PROGRAM Module_Status
VAR
	BLINK_Check		: Blink;
	BLINK_Module	: Blink;
	Index			: INT;
	TimerModule		: ARRAY [1..10] OF TOF;
	Ethercat_Status : ARRAY [1..10] OF Ethercat_status;
	FB_SystemData	: SystemData;
	FB_CpuUsage		: TC_CpuUsage;
	FB_SysLatency	: TC_SysLatency;
	FB_UPS			: FB_S_UPS_CX51x0;
END_VAR

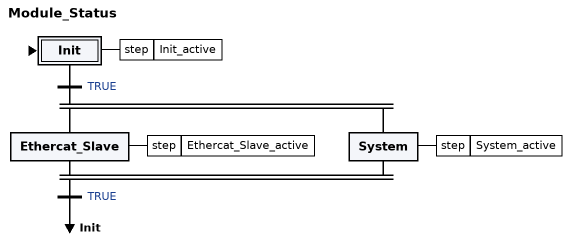
INITIAL_STEP Init:
    Init_active(N);  // step action
END_STEP
TRANSITION FROM Init TO (Ethercat_Slave, System)
    := TRUE;
END_TRANSITION
STEP Ethercat_Slave:
    Ethercat_Slave_active(N);  // step action
END_STEP
STEP System:
    System_active(N);  // step action
END_STEP
TRANSITION FROM (Ethercat_Slave, System) TO Init
    := TRUE;
END_TRANSITION

ACTION Ethercat_Slave_active:
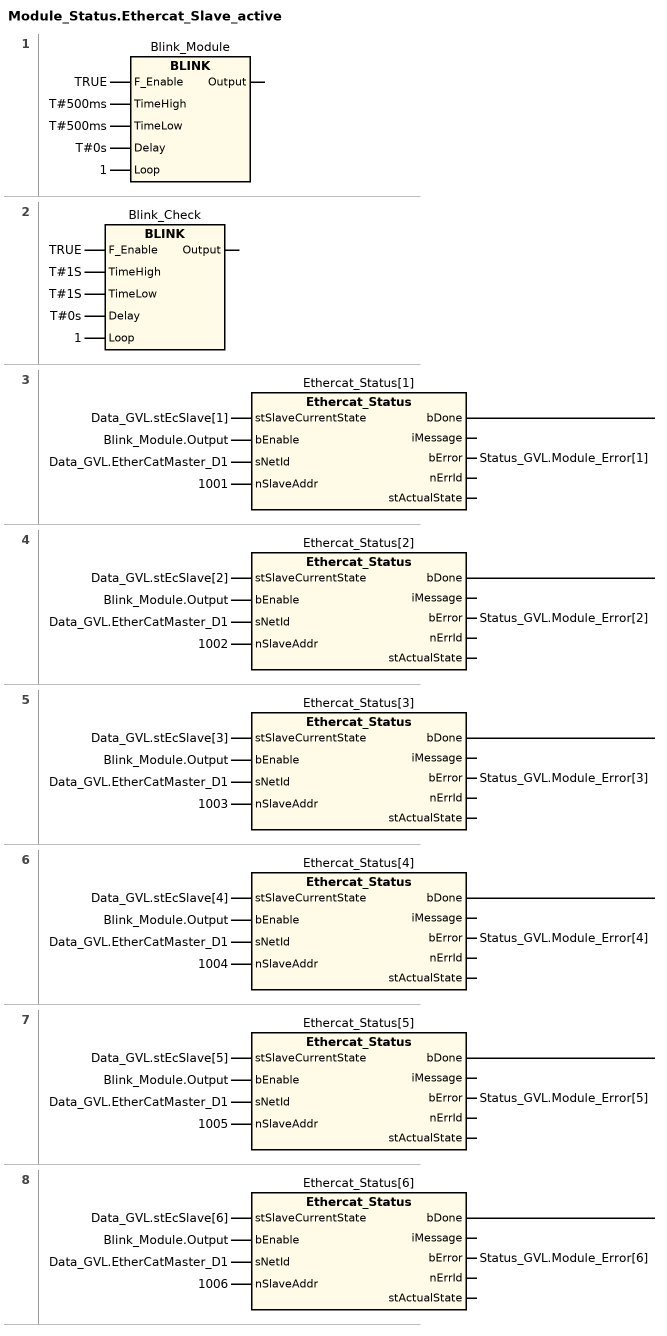
// NETWORK 1
Blink_Module(F_Enable := TRUE, TimeHigh := T#500ms, TimeLow := T#500ms, Delay := T#0s, Loop := 1); // BLINK

// NETWORK 2
Blink_Check(F_Enable := TRUE, TimeHigh := T#1S, TimeLow := T#1S, Delay := T#0s, Loop := 1); // BLINK

// NETWORK 3
Ethercat_Status[1](
    stSlaveCurrentState := Data_GVL.stEcSlave[1],
    bEnable := Blink_Module.Output,
    sNetId := Data_GVL.EtherCatMaster_D1,
    nSlaveAddr := 1001,
    bError => Status_GVL.Module_Error[1]); // Ethercat_Status

// NETWORK 4
Ethercat_Status[2](
    stSlaveCurrentState := Data_GVL.stEcSlave[2],
    bEnable := Blink_Module.Output,
    sNetId := Data_GVL.EtherCatMaster_D1,
    nSlaveAddr := 1002,
    bError => Status_GVL.Module_Error[2]); // Ethercat_Status

// NETWORK 5
Ethercat_Status[3](
    stSlaveCurrentState := Data_GVL.stEcSlave[3],
    bEnable := Blink_Module.Output,
    sNetId := Data_GVL.EtherCatMaster_D1,
    nSlaveAddr := 1003,
    bError => Status_GVL.Module_Error[3]); // Ethercat_Status

// NETWORK 6
Ethercat_Status[4](
    stSlaveCurrentState := Data_GVL.stEcSlave[4],
    bEnable := Blink_Module.Output,
    sNetId := Data_GVL.EtherCatMaster_D1,
    nSlaveAddr := 1004,
    bError => Status_GVL.Module_Error[4]); // Ethercat_Status

// NETWORK 7
Ethercat_Status[5](
    stSlaveCurrentState := Data_GVL.stEcSlave[5],
    bEnable := Blink_Module.Output,
    sNetId := Data_GVL.EtherCatMaster_D1,
    nSlaveAddr := 1005,
    bError => Status_GVL.Module_Error[5]); // Ethercat_Status

// NETWORK 8
Ethercat_Status[6](
    stSlaveCurrentState := Data_GVL.stEcSlave[6],
    bEnable := Blink_Module.Output,
    sNetId := Data_GVL.EtherCatMaster_D1,
    nSlaveAddr := 1006,
    bError => Status_GVL.Module_Error[6]); // Ethercat_Status

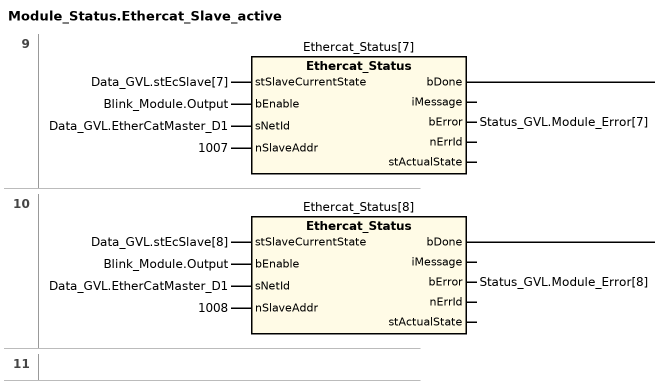
// NETWORK 9
Ethercat_Status[7](
    stSlaveCurrentState := Data_GVL.stEcSlave[7],
    bEnable := Blink_Module.Output,
    sNetId := Data_GVL.EtherCatMaster_D1,
    nSlaveAddr := 1007,
    bError => Status_GVL.Module_Error[7]); // Ethercat_Status

// NETWORK 10
Ethercat_Status[8](
    stSlaveCurrentState := Data_GVL.stEcSlave[8],
    bEnable := Blink_Module.Output,
    sNetId := Data_GVL.EtherCatMaster_D1,
    nSlaveAddr := 1008,
    bError => Status_GVL.Module_Error[8]); // Ethercat_Status

// NETWORK 11
END_ACTION

ACTION Init_active:
IF Blink_Check.Output THEN
	FOR Index := 1 TO 10 BY 1 DO
		TimerModule[Index](In:= Data_GVL.stEcSlave[Index].OP, PT:= T#2S);
		IF NOT TimerModule[Index].Q THEN 
			HMI_GVL.xOut_HMI_Status_EcSlave[Index] := FALSE;
		ELSE 
			HMI_GVL.xOut_HMI_Status_EcSlave[Index] := TRUE;
		END_IF
		
	END_FOR
ELSE
	Index := 1;
END_IF
END_ACTION

ACTION System_active:
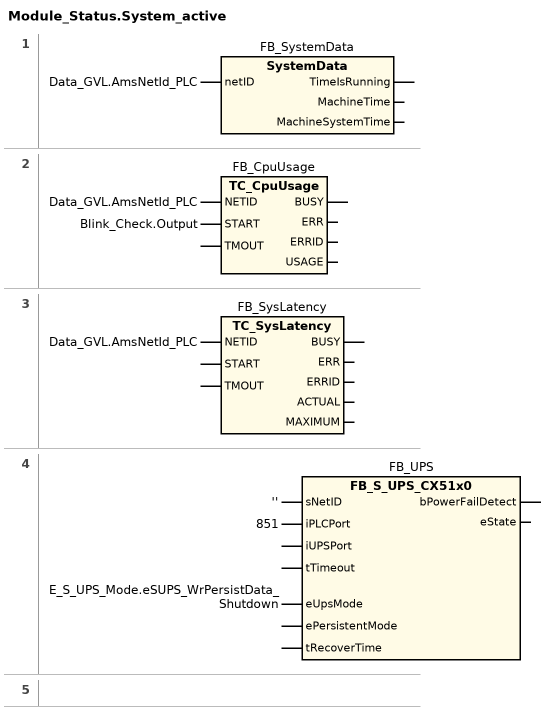
// NETWORK 1
FB_SystemData(netID := Data_GVL.AmsNetId_PLC); // SystemData

// NETWORK 2
FB_CpuUsage(NETID := Data_GVL.AmsNetId_PLC, START := Blink_Check.Output); // TC_CpuUsage

// NETWORK 3
FB_SysLatency(NETID := Data_GVL.AmsNetId_PLC); // TC_SysLatency

// NETWORK 4
FB_UPS(sNetID := '', iPLCPort := 851, eUpsMode := E_S_UPS_Mode.eSUPS_WrPersistData_Shutdown); // FB_S_UPS_CX51x0

// NETWORK 5
END_ACTION

END_PROGRAM

(* stored: Version 1.1.0.1, ProductVersion 3.1.4024.12
   POU Module_Status: Id {8029f611-6ea3-407c-a3cb-c97c2153bc88}, SpecialFunc None
   Action Ethercat_Slave_active: Id {57487703-7880-4487-b39b-2f5f3a8d13d7}
   Action Init_active: Id {5217ff6a-e1ac-4aa9-a4cd-23640febb78c}
   Action System_active: Id {0af128f1-724c-4108-9e31-8ae48e7b1e9c} *)
